# EPICS substitutions: xrmSlice/xrmSliceApp/Db/xrmSliceAI_PM_32CH.substitutions
file "xrmSliceAI_HT.template"
{
#Python 3.14.4 (main, Apr 16 2026, 00:00:00) [GCC 15.2.1 20260123 (Red Hat 15.2.1-7)] on linux
#Type "help", "copyright", "credits" or "license" for more information.
#>> for addr in range (0,32):
#...     print(f"        {{ {addr+1:02d}, {addr} }}")
#...
pattern { CH, ADDR }
        { 01, 0 }
        { 02, 1 }
        { 03, 2 }
        { 04, 3 }
        { 05, 4 }
        { 06, 5 }
        { 07, 6 }
        { 08, 7 }
        { 09, 8 }
        { 10, 9 }
        { 11, 10 }
        { 12, 11 }
        { 13, 12 }
        { 14, 13 }
        { 15, 14 }
        { 16, 15 }
        { 17, 16 }
        { 18, 17 }
        { 19, 18 }
        { 20, 19 }
        { 21, 20 }
        { 22, 21 }
        { 23, 22 }
        { 24, 23 }
        { 25, 24 }
        { 26, 25 }
        { 27, 26 }
        { 28, 27 }
        { 29, 28 }
        { 30, 29 }
        { 31, 30 }
        { 32, 31 }
}
